FUNCTION newMessage : BOOL
VAR_INPUT
	first: IncomingMessage;
	second: IncomingMessage;
END_VAR
VAR
END_VAR

newMessage := (first.id.dtime <> second.id.dtime)
	OR (first.id.ipv4 <> second.id.ipv4)
	OR (first.id.pid <> second.id.pid)
    OR (first.id.sequence <> second.id.sequence);

END_FUNCTION

(* stored: Version 1.1.0.1, ProductVersion 3.1.4022.12
   POU newMessage: Id {1e2a1f0a-e6df-4059-9106-13397bceb00c}, SpecialFunc None *)
